// TIA Portal V20 export
DATA_BLOCK "ConfigurationParameters_DB"   // DB32
AUTHOR : Siemens AG
FAMILY : ServiceControl
VERSION : 1.0
// stored: InstanceOfName ConfigurationParameters, InstanceOfType FB
"ConfigurationParameters"
   // VAR
   //    MTPAnalog { S7_SetPoint := 'True'} : Array[0..0] of "UDT_MTP_AnaServParam";
   //    MTPDigital { S7_SetPoint := 'True'} : Array[0..0] of "UDT_MTP_DIntServParam";
   //    MTPBinary { S7_SetPoint := 'True'} : Array[0..0] of "UDT_MTP_BinServParam";
   //    MTPString { S7_SetPoint := 'True'} : Array[0..0] of "UDT_MTP_StringServParam";
   // END_VAR
BEGIN
END_DATA_BLOCK
